(*
SPDX-FileCopyrightText: Â© 2026 Oleksandr Tiutyk <trofimich@gmail.com>
SPDX-License-Identifier: MIT
License: https://opensource.org/license/mit
*)

(*!
<summary>Encapsulates and decodes Beckhoff 16-bit EtherCAT analog input status word.</summary>
<description>
Provides decoded boolean properties for Underrange (bit 0), Overrange (bit 1), Limit 1 (bits 2..3),
Limit 2 (bits 4..5), Error (bit 6), TxPDO State (bit 14), and TxPDO Toggle (bit 15).
</description>
*)

FUNCTION_BLOCK ANALOG_INPUT_STATUS
VAR
	_Status : WORD;
END_VAR

(*!
<summary>Bit 6: General measurement or hardware error flag.</summary>
*)
{attribute 'monitoring' := 'call'}
PROPERTY FINAL Error : BOOL
GET
Error := _Status.6;
END_GET
END_PROPERTY

(*!
<summary>Bit 1: Upper limit of nominal measuring range exceeded.</summary>
*)
{attribute 'monitoring' := 'call'}
PROPERTY FINAL Overrange : BOOL
GET
Overrange := _Status.1;
END_GET
END_PROPERTY

(*!
<summary>Updates internal raw 16-bit status word.</summary>
<param name="status">Raw 16-bit EtherCAT channel status word.</param>
*)
METHOD SetStatus
VAR_INPUT
	status : WORD;
END_VAR
_Status := status;
END_METHOD

(*!
<summary>Bit 14: TxPDO data validity (0: valid, 1: invalid / bus error).</summary>
*)
{attribute 'monitoring' := 'call'}
PROPERTY FINAL TxPDOState : BOOL
GET
TxPDOState := _Status.14;
END_GET
END_PROPERTY

(*!
<summary>Bit 15: TxPDO communication toggle bit.</summary>
*)
{attribute 'monitoring' := 'call'}
PROPERTY FINAL TxPDOToggle : BOOL
GET
TxPDOToggle := _Status.15;
END_GET
END_PROPERTY

(*!
<summary>Bit 0: Lower limit of calibrated measuring range fallen below.</summary>
*)
{attribute 'monitoring' := 'call'}
PROPERTY FINAL Underrange : BOOL
GET
Underrange := _Status.0;
END_GET
END_PROPERTY

(*!
<summary>Bit 3: Input value is greater than or equal to Limit 1 threshold.</summary>
*)
{attribute 'monitoring' := 'call'}
PROPERTY FINAL ValueBiggerOrEqualLimit1 : BOOL
GET
ValueBiggerOrEqualLimit1 := _Status.3;
END_GET
END_PROPERTY

(*!
<summary>Bit 5: Input value is greater than or equal to Limit 2 threshold.</summary>
*)
{attribute 'monitoring' := 'call'}
PROPERTY FINAL ValueBiggerOrEqualLimit2 : BOOL
GET
ValueBiggerOrEqualLimit2 := _Status.5;
END_GET
END_PROPERTY

(*!
<summary>Bit 2: Input value is smaller than or equal to Limit 1 threshold.</summary>
*)
{attribute 'monitoring' := 'call'}
PROPERTY FINAL ValueSmallerOrEqualLimit1 : BOOL
GET
ValueSmallerOrEqualLimit1 := _Status.2;
END_GET
END_PROPERTY

(*!
<summary>Bit 4: Input value is smaller than or equal to Limit 2 threshold.</summary>
*)
{attribute 'monitoring' := 'call'}
PROPERTY FINAL ValueSmallerOrEqualLimit2 : BOOL
GET
ValueSmallerOrEqualLimit2 := _Status.4;
END_GET
END_PROPERTY

END_FUNCTION_BLOCK

(* stored: Version 1.1.0.1
   POU ANALOG_INPUT_STATUS: Id {c3761184-77be-4e03-8ba2-39b9618bad63}, SpecialFunc None
   Property Error: Id {7c14b191-91fd-4588-b67e-152ef5775adb}
   Get Get: Id {7c6a5d0f-e45b-426a-96bb-16e52fdf107d}
   Property Overrange: Id {1bd71454-ce03-40c9-b9ff-7f392a5a4464}
   Get Get: Id {a7e18e48-4c97-4fdc-b7da-4937dcd6c517}
   Method SetStatus: Id {33141c99-8102-401e-8f13-439953bd0ad2}
   Property TxPDOState: Id {8ba45a8e-c734-43a4-a857-140efc9a069b}
   Get Get: Id {b587ce97-fea7-42a8-9823-497421797695}
   Property TxPDOToggle: Id {72f1f652-ed5c-4665-987b-fec1e74f1009}
   Get Get: Id {ec9d41ec-d81f-418e-bbd5-1923c72e40b2}
   Property Underrange: Id {94d26341-48fe-4af5-9bac-ba53b413d45f}
   Get Get: Id {8580446d-3b45-4524-9943-11fece3e42bd}
   Property ValueBiggerOrEqualLimit1: Id {60241d05-b62b-4928-a1b0-6d9c586e849c}
   Get Get: Id {02fd67d6-7b5c-447a-9326-401d4f7904e5}
   Property ValueBiggerOrEqualLimit2: Id {a618c40b-e461-4edf-8aa6-54c2a36a5897}
   Get Get: Id {5be5185a-52b7-4156-bdae-a3d42f19fb42}
   Property ValueSmallerOrEqualLimit1: Id {61e2653f-d07a-4700-8180-3acc5d85f0ad}
   Get Get: Id {39557e1e-71e5-4073-bb39-ce6fa6046d65}
   Property ValueSmallerOrEqualLimit2: Id {cf074ec1-302e-4ddb-979a-b16864ffddab}
   Get Get: Id {91b341a6-a274-4d48-974e-10a462c05eac} *)
